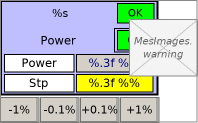
VISUALIZATION VISU_CANON  // 198x123
VAR_IN_OUT
	m_Input_SOURCE : BLOCK_SOURCE_JOULE;
END_VAR
    Rectangle (0,0 158x95)
    Rectangle (3,30 110x21), "Power"
    Rectangle (117,3 37x20), "NOK", invisible if: NOT m_Input_SOURCE.STATE_NOK
    Rectangle (117,30 37x20), "OFF", invisible if: m_Input_SOURCE.STATE_EJ_ON
    Rectangle (117,3 37x20), "OK", invisible if: m_Input_SOURCE.STATE_NOK
    Rectangle (117,30 37x20), "ON", invisible if: NOT m_Input_SOURCE.STATE_EJ_ON
    RoundedRectangle (4,54 70x18), "Power", invisible if: Global_Variables.MACHINE.State_manu
    RoundedRectangle (76,54 77x18), "%.3f %%", text variable: m_Input_SOURCE.STATE_POWER, invisible if: Global_Variables.MACHINE.State_manu
    Rectangle (0,3 120x21), "%s", text variable: m_Input_SOURCE.MNEMO
    Polyline (7,35)
    RoundedRectangle (4,74 70x18), "Stp", invisible if: NOT Global_Variables.PRG_USER.ACTU_USER.MAINTENANCE OR NOT MACHINE.State_manu
    RoundedRectangle (76,74 77x18), "%.3f %%", text variable: m_Input_SOURCE.PRM_POWER, invisible if: NOT Global_Variables.PRG_USER.ACTU_USER.MAINTENANCE OR NOT MACHINE.STATE_Manu
        OnMouseDown: write the text variable via InputWithLimits, min 0, max 100
    Rectangle (114,28 41x24), invisible if: NOT m_Input_SOURCE.EJ.AUTOR_ON_IHM AND NOT m_Input_SOURCE.EJ.AUTOR_Off_IHM, input disabled if: (NOT m_Input_SOURCE.EJ.AUTOR_ON_IHM AND NOT m_Input_SOURCE.EJ.AUTOR_OFF_IHM) OR NOT PRG_User.ACTU_USER.MAINTENANCE
        tap m_Input_SOURCE.EJ.M_On
    Image (129,19 69x57), invisible if: NOT m_Input_SOURCE.STATE_NOK, image: MesImages.warning
    Button (0,97 39x26), "-1%", invisible if: NOT Global_Variables.PRG_USER.ACTU_USER.MAINTENANCE OR NOT MACHINE.STATE_Manu OR (m_Input_SOURCE.PRM_POWER<1.0)
        OnMouseClick: execute { m_Input_SOURCE.PRM_POWER := m_Input_SOURCE.PRM_POWER - 1.0; }
    Button (40,97 39x26), "-0.1%", invisible if: NOT Global_Variables.PRG_USER.ACTU_USER.MAINTENANCE OR NOT MACHINE.STATE_Manu OR (m_Input_SOURCE.PRM_POWER<0.1)
        OnMouseClick: execute { m_Input_SOURCE.PRM_POWER := m_Input_SOURCE.PRM_POWER - 0.1; }
    Button (80,97 39x26), "+0.1%", invisible if: NOT Global_Variables.PRG_USER.ACTU_USER.MAINTENANCE OR NOT MACHINE.STATE_Manu OR (m_Input_SOURCE.PRM_POWER>99.9)
        OnMouseClick: execute { m_Input_SOURCE.PRM_POWER := m_Input_SOURCE.PRM_POWER + 0.1; }
    Button (120,97 39x26), "+1%", invisible if: NOT Global_Variables.PRG_USER.ACTU_USER.MAINTENANCE OR NOT MACHINE.STATE_Manu OR (m_Input_SOURCE.PRM_POWER>99.0)
        OnMouseClick: execute { m_Input_SOURCE.PRM_POWER := m_Input_SOURCE.PRM_POWER + 1.0; }
END_VISUALIZATION

// ---- Visualizations/Symbole/EVAP/VISU_CANON_GENIUS_ETH.TcVIS
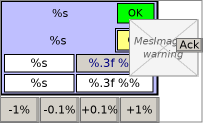
VISUALIZATION VISU_CANON_GENIUS_ETH  // 203x123
VAR_IN_OUT
	m_Input_SOURCE : BLOCK_SOURCE_GENIUS_ETHERCAT;
END_VAR
    Rectangle (0,0 158x95)
    Rectangle (3,30 110x21), "%s", text list: 'TextList_Evap', text index: 2
    Rectangle (117,3 37x20), "NOK", invisible if: NOT m_Input_SOURCE.STATE_NOK
    Rectangle (117,30 37x20), "OFF", invisible if: m_Input_SOURCE.STATE_SRC OR m_Input_SOURCE.STATE_SRC_ON
    Rectangle (117,3 37x20), "OK", invisible if: m_Input_SOURCE.STATE_NOK
    Rectangle (117,30 37x20), "ON", invisible if: NOT m_Input_SOURCE.STATE_SRC AND NOT m_Input_SOURCE.STATE_SRC_ON
    RoundedRectangle (4,54 70x18), "%s", invisible if: Global_Variables.MACHINE.State_manu, text list: 'TextList_Evap', text index: 4
    RoundedRectangle (76,54 77x18), "%.3f %%", text variable: m_Input_SOURCE.STATE_COURANT, invisible if: Global_Variables.MACHINE.State_manu
    Rectangle (117,30 37x20), "ON", invisible if: m_Input_SOURCE.STATE_SRC_ON OR NOT m_Input_SOURCE.STATE_SRC
    Rectangle (0,3 120x21), "%s", text variable: m_Input_SOURCE.MNEMO
    Polyline (7,35)
    RoundedRectangle (4,74 70x18), "%s", invisible if: NOT Global_Variables.PRG_USER.ACTU_USER.MAINTENANCE OR NOT MACHINE.State_manu, text list: 'TextList_Evap', text index: 4
    RoundedRectangle (76,74 77x18), "%.3f %%", text variable: m_Input_SOURCE.PRM_COURANT, invisible if: NOT Global_Variables.PRG_USER.ACTU_USER.MAINTENANCE OR NOT MACHINE.STATE_Manu
        OnMouseDown: write the text variable via VisuDialogs.Numpad, min 0, max 100
    Rectangle (115,28 41x24), invisible if: NOT m_Input_SOURCE.SRC.AUTOR_ON_IHM AND NOT m_Input_SOURCE.SRC.AUTOR_OFF_IHM, input disabled if: (NOT m_Input_SOURCE.SRC.AUTOR_ON_IHM AND NOT m_Input_SOURCE.SRC.AUTOR_OFF_IHM) OR NOT PRG_User.ACTU_USER.MAINTENANCE
        tap m_Input_SOURCE.SRC.M_On
    Image (129,19 69x57), invisible if: NOT m_Input_SOURCE.SRC.STATE_Nok AND NOT m_Input_SOURCE.DEF_Source.DEF AND NOT m_Input_SOURCE.DEF_Communication.DEF, image: MesImages.warning
    Button (0,97 39x26), "-1%", invisible if: NOT Global_Variables.PRG_USER.ACTU_USER.MAINTENANCE OR NOT MACHINE.STATE_Manu
        OnMouseClick: execute { m_Input_SOURCE.PRM_COURANT := m_Input_SOURCE.PRM_COURANT - 1; }
    Button (40,97 39x26), "-0.1%", invisible if: NOT Global_Variables.PRG_USER.ACTU_USER.MAINTENANCE OR NOT MACHINE.STATE_Manu
        OnMouseClick: execute { m_Input_SOURCE.PRM_COURANT := m_Input_SOURCE.PRM_COURANT - 0.1; }
    Button (80,97 39x26), "+0.1%", invisible if: NOT Global_Variables.PRG_USER.ACTU_USER.MAINTENANCE OR NOT MACHINE.STATE_Manu
        OnMouseClick: execute { m_Input_SOURCE.PRM_COURANT := m_Input_SOURCE.PRM_COURANT + 0.1; }
    Button (120,97 39x26), "+1%", invisible if: NOT Global_Variables.PRG_USER.ACTU_USER.MAINTENANCE OR NOT MACHINE.STATE_Manu
        OnMouseClick: execute { m_Input_SOURCE.PRM_COURANT := m_Input_SOURCE.PRM_COURANT + 1; }
    Button (176,38 27x14), "Ack", invisible if: NOT m_Input_SOURCE.HV.STATE_Nok AND NOT m_Input_SOURCE.DEF_Source.DEF AND NOT m_Input_SOURCE.DEF_Communication.DEF AND NOT m_Input_SOURCE.DEF_HV.DEF
        tap m_Input_SOURCE.M_Ack
END_VISUALIZATION

// ---- Visualizations/Symbole/EVAP/VISU_CANON_ST10.TcVIS
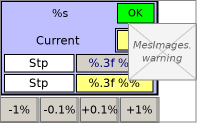
VISUALIZATION VISU_CANON_ST10  // 197x123
VAR_IN_OUT
	m_Input_SOURCE : BLOCK_CANON_ST10;
END_VAR
    Rectangle (0,0 158x95)
    Rectangle (3,30 110x21), "Current"
    Rectangle (117,3 37x20), "NOK", invisible if: NOT m_Input_SOURCE.STATE_NOK
    Rectangle (117,30 37x20), "OFF", invisible if: m_Input_SOURCE.STATE_SRC OR m_Input_SOURCE.STATE_SRC_ON
    Rectangle (117,3 37x20), "OK", invisible if: m_Input_SOURCE.STATE_NOK
    Rectangle (117,30 37x20), "ON", invisible if: NOT m_Input_SOURCE.STATE_SRC AND NOT m_Input_SOURCE.STATE_SRC_ON
    RoundedRectangle (4,54 70x18), "Stp", invisible if: Global_Variables.MACHINE.State_manu
    RoundedRectangle (76,54 77x18), "%.3f %%", text variable: m_Input_SOURCE.AO_QIEM.Value, invisible if: Global_Variables.MACHINE.State_manu
    Rectangle (117,30 37x20), "ON", invisible if: m_Input_SOURCE.STATE_SRC_ON OR Not m_Input_SOURCE.STATE_SRC
    Rectangle (0,3 120x21), "%s", text variable: m_Input_SOURCE.MNEMO
    Polyline (7,35)
    RoundedRectangle (4,74 70x18), "Stp", invisible if: NOT Global_Variables.PRG_USER.ACTU_USER.MAINTENANCE OR NOT MACHINE.State_manu
    RoundedRectangle (76,74 77x18), "%.3f %%", text variable: m_Input_SOURCE.PRM_COURANT, invisible if: NOT Global_Variables.PRG_USER.ACTU_USER.MAINTENANCE OR NOT MACHINE.STATE_Manu
        OnMouseDown: write the text variable via InputWithLimits, min 0, max 100
    Rectangle (115,28 41x24), invisible if: NOT m_Input_SOURCE.SRC.AUTOR_ON_IHM AND NOT m_Input_SOURCE.SRC.AUTOR_OFF_IHM, input disabled if: (NOT m_Input_SOURCE.SRC.AUTOR_ON_IHM AND NOT m_Input_SOURCE.SRC.AUTOR_OFF_IHM) OR NOT PRG_User.ACTU_USER.MAINTENANCE
        tap m_Input_SOURCE.SRC.M_On
    Image (128,23 69x57), invisible if: NOT m_Input_SOURCE.STATE_NOK, image: MesImages.warning
    Button (0,97 39x26), "-1%", invisible if: NOT Global_Variables.PRG_USER.ACTU_USER.MAINTENANCE OR NOT MACHINE.STATE_Manu OR (m_Input_SOURCE.PRM_COURANT<1.0)
        OnMouseClick: execute { m_Input_SOURCE.PRM_COURANT := m_Input_SOURCE.PRM_COURANT - 1.0; }
    Button (40,97 39x26), "-0.1%", invisible if: NOT Global_Variables.PRG_USER.ACTU_USER.MAINTENANCE OR NOT MACHINE.STATE_Manu OR (m_Input_SOURCE.PRM_COURANT<0.1)
        OnMouseClick: execute { m_Input_SOURCE.PRM_COURANT := m_Input_SOURCE.PRM_COURANT - 0.1; }
    Button (80,97 39x26), "+0.1%", invisible if: NOT Global_Variables.PRG_USER.ACTU_USER.MAINTENANCE OR NOT MACHINE.STATE_Manu OR (m_Input_SOURCE.PRM_COURANT>99.9)
        OnMouseClick: execute { m_Input_SOURCE.PRM_COURANT := m_Input_SOURCE.PRM_COURANT + 0.1; }
    Button (120,97 39x26), "+1%", invisible if: NOT Global_Variables.PRG_USER.ACTU_USER.MAINTENANCE OR NOT MACHINE.STATE_Manu OR (m_Input_SOURCE.PRM_COURANT>99.0)
        OnMouseClick: execute { m_Input_SOURCE.PRM_COURANT := m_Input_SOURCE.PRM_COURANT + 1.0; }
END_VISUALIZATION

// ---- Visualizations/Symbole/EVAP/VISU_CONF_BAL.TcVIS
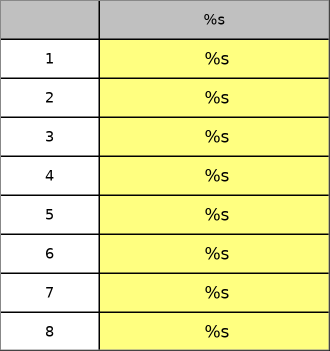
VISUALIZATION VISU_CONF_BAL  // 330x351
VAR_IN_OUT
	m_Input_SWEEP : BLOCK_TELEMARK_CHEETAH_SWEEP;
END_VAR
    Rectangle (0,0 99x39)
    Rectangle (99,39 231x39), "%s", text variable: m_Input_SWEEP.PRM_BAL[1], input disabled if: NOT Global_Variables.PRG_USER.ACTU_USER.CONF_MACHINE
        OnMouseDown: write the text variable via InputWithLimits
    Rectangle (99,0 231x39), "%s", text list: 'TextList_Config_Evap', text index: 8
    Rectangle (0,39 99x39), "1"
    Rectangle (0,78 99x39), "2"
    Rectangle (99,78 231x39), "%s", text variable: m_Input_SWEEP.PRM_BAL[2], input disabled if: NOT Global_Variables.PRG_USER.ACTU_USER.CONF_MACHINE
        OnMouseDown: write the text variable via InputWithLimits
    Rectangle (0,117 99x39), "3"
    Rectangle (99,117 231x39), "%s", text variable: m_Input_SWEEP.PRM_BAL[3], input disabled if: NOT Global_Variables.PRG_USER.ACTU_USER.CONF_MACHINE
        OnMouseDown: write the text variable via InputWithLimits
    Rectangle (0,156 99x39), "4"
    Rectangle (99,156 231x39), "%s", text variable: m_Input_SWEEP.PRM_BAL[4], input disabled if: NOT Global_Variables.PRG_USER.ACTU_USER.CONF_MACHINE
        OnMouseDown: write the text variable via InputWithLimits
    Rectangle (99,195 231x39), "%s", text variable: m_Input_SWEEP.PRM_BAL[5], input disabled if: NOT Global_Variables.PRG_USER.ACTU_USER.CONF_MACHINE
        OnMouseDown: write the text variable via InputWithLimits
    Rectangle (0,195 99x39), "5"
    Rectangle (0,234 99x39), "6"
    Rectangle (99,234 231x39), "%s", text variable: m_Input_SWEEP.PRM_BAL[6], input disabled if: NOT Global_Variables.PRG_USER.ACTU_USER.CONF_MACHINE
        OnMouseDown: write the text variable via InputWithLimits
    Rectangle (0,273 99x39), "7"
    Rectangle (99,273 231x39), "%s", text variable: m_Input_SWEEP.PRM_BAL[7], input disabled if: NOT Global_Variables.PRG_USER.ACTU_USER.CONF_MACHINE
        OnMouseDown: write the text variable via InputWithLimits
    Rectangle (0,312 99x39), "8"
    Rectangle (99,312 231x39), "%s", text variable: m_Input_SWEEP.PRM_BAL[8], input disabled if: NOT Global_Variables.PRG_USER.ACTU_USER.CONF_MACHINE
        OnMouseDown: write the text variable via InputWithLimits
END_VISUALIZATION

// ---- Visualizations/Symbole/EVAP/VISU_CONF_MAT.TcVIS
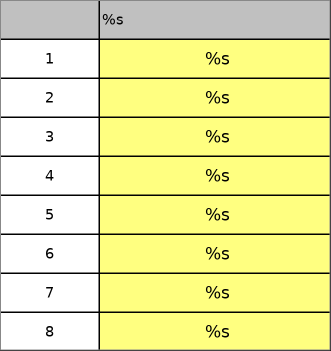
VISUALIZATION VISU_CONF_MAT  // 331x351
VAR_IN_OUT
	m_Input_CRUCIBLE : BLOCK_IND_CR_396_TELEMARK;
END_VAR
    Rectangle (0,0 99x39)
    Rectangle (99,39 232x39), "%s", text variable: m_Input_CRUCIBLE.PRM_MAT[1], input disabled if: NOT Global_Variables.PRG_USER.ACTU_USER.CONF_MACHINE
        OnMouseDown: write the text variable via InputWithLimits
    Rectangle (99,0 232x39), "%s", text list: 'TextList_Config_Evap', text index: 7
    Rectangle (0,39 99x39), "1"
    Rectangle (0,78 99x39), "2", invisible if: m_Input_CRUCIBLE.CONF_NCR <2
    Rectangle (99,78 232x39), "%s", text variable: m_Input_CRUCIBLE.PRM_MAT[2], invisible if: m_Input_CRUCIBLE.CONF_NCR <2, input disabled if: NOT Global_Variables.PRG_USER.ACTU_USER.CONF_MACHINE
        OnMouseDown: write the text variable via InputWithLimits
    Rectangle (0,117 99x39), "3", invisible if: m_Input_CRUCIBLE.CONF_NCR <3
    Rectangle (99,117 232x39), "%s", text variable: m_Input_CRUCIBLE.PRM_MAT[3], invisible if: m_Input_CRUCIBLE.CONF_NCR <3, input disabled if: NOT Global_Variables.PRG_USER.ACTU_USER.CONF_MACHINE
        OnMouseDown: write the text variable via InputWithLimits
    Rectangle (0,156 99x39), "4", invisible if: m_Input_CRUCIBLE.CONF_NCR <4
    Rectangle (99,156 232x39), "%s", text variable: m_Input_CRUCIBLE.PRM_MAT[4], invisible if: m_Input_CRUCIBLE.CONF_NCR <4, input disabled if: NOT Global_Variables.PRG_USER.ACTU_USER.CONF_MACHINE
        OnMouseDown: write the text variable via InputWithLimits
    Rectangle (0,195 99x39), "5", invisible if: m_Input_CRUCIBLE.CONF_NCR <5
    Rectangle (99,195 232x39), "%s", text variable: m_Input_CRUCIBLE.PRM_MAT[5], invisible if: m_Input_CRUCIBLE.CONF_NCR <5, input disabled if: NOT Global_Variables.PRG_USER.ACTU_USER.CONF_MACHINE
        OnMouseDown: write the text variable via InputWithLimits
    Rectangle (0,234 99x39), "6", invisible if: m_Input_CRUCIBLE.CONF_NCR <6
    Rectangle (99,234 232x39), "%s", text variable: m_Input_CRUCIBLE.PRM_MAT[6], invisible if: m_Input_CRUCIBLE.CONF_NCR <6, input disabled if: NOT Global_Variables.PRG_USER.ACTU_USER.CONF_MACHINE
        OnMouseDown: write the text variable via InputWithLimits
    Rectangle (0,273 99x39), "7", invisible if: m_Input_CRUCIBLE.CONF_NCR <7
    Rectangle (99,273 232x39), "%s", text variable: m_Input_CRUCIBLE.PRM_MAT[7], invisible if: m_Input_CRUCIBLE.CONF_NCR <7, input disabled if: NOT Global_Variables.PRG_USER.ACTU_USER.CONF_MACHINE
        OnMouseDown: write the text variable via InputWithLimits
    Rectangle (0,312 99x39), "8", invisible if: m_Input_CRUCIBLE.CONF_NCR <8
    Rectangle (99,312 232x39), "%s", text variable: m_Input_CRUCIBLE.PRM_MAT[8], invisible if: m_Input_CRUCIBLE.CONF_NCR <8, input disabled if: NOT Global_Variables.PRG_USER.ACTU_USER.CONF_MACHINE
        OnMouseDown: write the text variable via InputWithLimits
END_VISUALIZATION

// ---- Visualizations/Symbole/EVAP/VISU_CREUSET_old.TcVIS
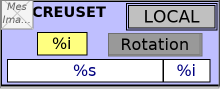
VISUALIZATION VISU_CREUSET_old  // 220x89
VAR_IN_OUT
	m_Input_CREUSET : BLOCK_IND_CR_379_TELEMARK;
END_VAR
    Rectangle (0,0 220x86)
    RoundedRectangle (37,32 50x23), "%i", text variable: m_Input_CREUSET.PRM_NCR, invisible if: NOT Global_Variables.PRG_USER.ACTU_USER.MAINTENANCE OR NOT MACHINE.State_manu
        OnMouseDown: write the text variable via InputWithLimits, min 1, max m_Input_CREUSET.CONF_NCR
    Rectangle (6,3 126x18), "CREUSET"
    RoundedRectangle (7,59 156x23), "%s", text variable: m_Input_CREUSET.STATE_MAT
    RoundedRectangle (163,59 47x23), "%i", text variable: m_Input_CREUSET.STATE_POS
    Button (108,33 94x23), "Rotation", invisible if: NOT m_Input_CREUSET.AUTOR_Change_IHM OR NOT PRG_User.ACTU_USER.MAINTENANCE
        tap m_Input_CREUSET.M_Change
    Image (1,-3 32x32), invisible if: NOT m_Input_CREUSET.State_nok, image: MesImages.warning
    RoundedRectangle (128,5 87x23), "REMOTE", invisible if: not m_Input_CREUSET.OUT_RMT
    RoundedRectangle (128,5 87x23), "LOCAL", invisible if: m_Input_CREUSET.OUT_RMT
    Rectangle (126,3 91x27), invisible if: Not m_Input_CREUSET.AUTOR_Remote_IHM, input disabled if: NOT PRG_User.ACTU_USER.MAINTENANCE
        tap m_Input_CREUSET.M_Remote
END_VISUALIZATION

// ---- Visualizations/Symbole/EVAP/VISU_CREUSET.TcVIS
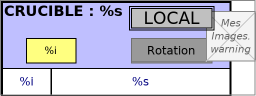
VISUALIZATION VISU_CREUSET  // 256x96
VAR_IN_OUT
	m_Input_CREUSET : BLOCK_IND_CR_396_TELEMARK;
END_VAR
VAR_INPUT
	m_Input_NUM_CRUCIBLE : SINT;
END_VAR
    Rectangle (1,1 230x95), "CRUCIBLE : %s", text variable: m_Input_NUM_CRUCIBLE
    RoundedRectangle (26,38 50x25), "%i", text variable: m_Input_CREUSET.PRM_NCR, invisible if: NOT Global_Variables.PRG_USER.ACTU_USER.MAINTENANCE OR NOT MACHINE.State_manu
        OnMouseDown: write the text variable via InputWithLimits, min 1, max 6
    Rectangle (51,68 179x27), "%s", text variable: m_Input_CREUSET.STATE_MAT
    Rectangle (2,68 49x27), "%i", text variable: m_Input_CREUSET.STATE_POS
    Button (131,38 81x25), "Rotation", colour toggle: m_Input_CREUSET.STATE_ROT, invisible if: NOT m_Input_CREUSET.AUTOR_Change_IHM OR NOT PRG_User.ACTU_USER.MAINTENANCE
        tap m_Input_CREUSET.M_Change
    Image (206,11 50x50), invisible if: NOT m_Input_CREUSET.State_nok, image: MesImages.warning
    RoundedRectangle (131,8 81x20), "REMOTE", invisible if: not m_Input_CREUSET.OUT_RMT
    RoundedRectangle (131,8 81x20), "LOCAL", invisible if: m_Input_CREUSET.OUT_RMT
    Rectangle (129,6 85x24), invisible if: Not m_Input_CREUSET.AUTOR_Remote_IHM, input disabled if: NOT PRG_User.ACTU_USER.MAINTENANCE
        tap m_Input_CREUSET.M_Remote
END_VISUALIZATION

// ---- Visualizations/Symbole/EVAP/VISU_CREUSET_V3.TcVIS
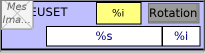
VISUALIZATION VISU_CREUSET_V3  // 205x53
VAR_IN_OUT
	m_Input_CREUSET : BLOCK_IND_CR_379_TELEMARK_V3;
END_VAR
    Rectangle (0,0 205x50)
    RoundedRectangle (96,2 45x22), "%i", text variable: m_Input_CREUSET.PRM_NCR, invisible if: NOT Global_Variables.PRG_USER.ACTU_USER.MAINTENANCE OR NOT MACHINE.State_manu
        OnMouseDown: write the text variable via InputWithLimits
    Rectangle (0,3 81x18), "CREUSET"
    Rectangle (1,26 48x18), text list: 'TextList_Evap', text index: 5
    RoundedRectangle (46,26 116x20), "%s", text variable: m_Input_CREUSET.STATE_MAT
    RoundedRectangle (162,26 38x20), "%i", text variable: m_Input_CREUSET.STATE_POS
    Button (148,3 51x20), "Rotation", invisible if: NOT m_Input_CREUSET.AUTOR_Change_IHM OR NOT PRG_User.ACTU_USER.MAINTENANCE
        tap m_Input_CREUSET.M_Change
    Image (1,-3 32x32), invisible if: NOT m_Input_CREUSET.State_nok, image: MesImages.warning
END_VISUALIZATION

// ---- Visualizations/Symbole/EVAP/VISU_CR_SW_GENIUS_ETH.TcVIS
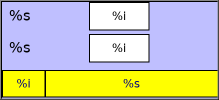
VISUALIZATION VISU_CR_SW_GENIUS_ETH  // 219x100
VAR_IN_OUT
	m_Input_BALAYAGE : BLOCK_IND_CREUSET_GENIUS_ETHERCAT;
END_VAR
    Rectangle (0,0 219x100)
    Rectangle (6,1 118x29), "%s", text list: 'TextList_Evap', text index: 0
    Rectangle (2,70 43x27), "%i", text variable: m_Input_BALAYAGE.STATE_POS_CR
    Rectangle (45,70 173x27), "%s", text variable: m_Input_BALAYAGE.STATE_MAT
    RoundedRectangle (89,2 60x28), "%i", text variable: m_Input_BALAYAGE.PRM_NCR, input disabled if: NOT Global_Variables.PRG_USER.ACTU_USER.MAINTENANCE OR NOT MACHINE.STATE_Manu
        OnMouseDown: write the text variable via VisuDialogs.Numpad, min 1, max m_Input_BALAYAGE.CONF_NCR
    Rectangle (6,33 118x29), "%s", text list: 'TextList_Evap', text index: 1
    RoundedRectangle (89,34 60x28), "%i", text variable: m_Input_BALAYAGE.PRM_NBAL, input disabled if: NOT Global_Variables.PRG_USER.ACTU_USER.MAINTENANCE OR NOT MACHINE.STATE_Manu
        OnMouseDown: write the text variable via VisuDialogs.Numpad, min 1, max 8
END_VISUALIZATION

// ---- Visualizations/Symbole/EVAP/VISU_HT_CANON_ST10.TcVIS
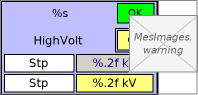
VISUALIZATION VISU_HT_CANON_ST10  // 198x95
VAR_IN_OUT
	m_Input_SOURCE : BLOCK_CANON_ST10;
END_VAR
    Rectangle (0,0 158x95)
    Rectangle (3,30 110x21), "HighVolt"
    Rectangle (117,3 37x20), "NOK", invisible if: NOT m_Input_SOURCE.STATE_NOK
    Rectangle (117,30 37x20), "OFF", invisible if: m_Input_SOURCE.STATE_HV OR m_Input_SOURCE.STATE_HV_ON
    Rectangle (117,3 37x20), "OK", invisible if: m_Input_SOURCE.STATE_NOK
    Rectangle (117,30 37x20), "ON", invisible if: NOT m_Input_SOURCE.STATE_HV AND NOT m_Input_SOURCE.STATE_HV_ON
    RoundedRectangle (4,54 70x18), "Stp", invisible if: Global_Variables.MACHINE.State_manu
    RoundedRectangle (76,54 77x18), "%.2f kV", text variable: m_Input_SOURCE.AO_QUHV.Value, invisible if: Global_Variables.MACHINE.State_manu
    Rectangle (117,30 37x20), "ON", invisible if: m_Input_SOURCE.STATE_HV_ON OR NOT m_Input_SOURCE.STATE_HV
    Rectangle (0,3 120x21), "%s", text variable: m_Input_SOURCE.MNEMO
    Polyline (7,35)
    RoundedRectangle (4,74 70x18), "Stp", invisible if: NOT Global_Variables.PRG_USER.ACTU_USER.MAINTENANCE OR NOT MACHINE.State_manu
    RoundedRectangle (76,74 77x18), "%.2f kV", text variable: m_Input_SOURCE.PRM_TENSION, invisible if: NOT Global_Variables.PRG_USER.ACTU_USER.MAINTENANCE OR NOT MACHINE.STATE_Manu
        OnMouseDown: write the text variable via InputWithLimits, min 7, max 10
    Rectangle (115,28 41x24), invisible if: NOT m_Input_SOURCE.HV.AUTOR_ON_IHM AND NOT m_Input_SOURCE.HV.AUTOR_OFF_IHM, input disabled if: (NOT m_Input_SOURCE.HV.AUTOR_ON_IHM AND NOT m_Input_SOURCE.HV.AUTOR_OFF_IHM) OR NOT PRG_User.ACTU_USER.MAINTENANCE
        tap m_Input_SOURCE.HV.M_On
    Image (129,15 69x57), invisible if: NOT m_Input_SOURCE.STATE_NOK, image: MesImages.warning
END_VISUALIZATION

// ---- Visualizations/Symbole/EVAP/VISU_HT_GENIUS_ETH.TcVIS
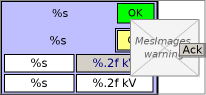
VISUALIZATION VISU_HT_GENIUS_ETH  // 206x95
VAR_IN_OUT
	m_Input_SOURCE : BLOCK_SOURCE_GENIUS_ETHERCAT;
END_VAR
    Rectangle (0,0 158x95)
    Rectangle (3,30 110x21), "%s", text list: 'TextList_Evap', text index: 3
    Rectangle (117,3 37x20), "NOK", invisible if: NOT m_Input_SOURCE.STATE_NOK
    Rectangle (117,30 37x20), "OFF", invisible if: m_Input_SOURCE.STATE_HV OR m_Input_SOURCE.STATE_HV_ON
    Rectangle (117,3 37x20), "OK", invisible if: m_Input_SOURCE.STATE_NOK
    Rectangle (117,30 37x20), "ON", invisible if: NOT m_Input_SOURCE.STATE_HV AND NOT m_Input_SOURCE.STATE_HV_ON
    RoundedRectangle (4,54 70x18), "%s", invisible if: Global_Variables.MACHINE.State_manu, text list: 'TextList_Evap', text index: 4
    RoundedRectangle (76,54 77x18), "%.2f kV", text variable: m_Input_SOURCE.STATE_TENSION, invisible if: Global_Variables.MACHINE.State_manu
    Rectangle (117,30 37x20), "ON", invisible if: m_Input_SOURCE.STATE_HV_ON OR NOT m_Input_SOURCE.STATE_HV
    Rectangle (0,3 120x21), "%s", text variable: m_Input_SOURCE.MNEMO
    Polyline (7,35)
    RoundedRectangle (4,74 70x18), "%s", invisible if: NOT Global_Variables.PRG_USER.ACTU_USER.MAINTENANCE OR NOT MACHINE.State_manu, text list: 'TextList_Evap', text index: 4
    RoundedRectangle (76,74 77x18), "%.2f kV", text variable: m_Input_SOURCE.PRM_TENSION, invisible if: NOT Global_Variables.PRG_USER.ACTU_USER.MAINTENANCE OR NOT MACHINE.STATE_Manu
        OnMouseDown: write the text variable via VisuDialogs.Numpad, min 7, max 10
    Rectangle (115,28 41x24), invisible if: NOT m_Input_SOURCE.HV.AUTOR_ON_IHM AND NOT m_Input_SOURCE.HV.AUTOR_OFF_IHM, input disabled if: (NOT m_Input_SOURCE.HV.AUTOR_ON_IHM AND NOT m_Input_SOURCE.HV.AUTOR_OFF_IHM) OR NOT PRG_User.ACTU_USER.MAINTENANCE
        tap m_Input_SOURCE.HV.M_On
    Image (130,19 69x57), invisible if: NOT m_Input_SOURCE.HV.STATE_Nok AND NOT m_Input_SOURCE.DEF_Source.DEF AND NOT m_Input_SOURCE.DEF_Communication.DEF AND NOT m_Input_SOURCE.DEF_HV.DEF, image: MesImages.warning
    Button (179,43 27x14), "Ack", invisible if: NOT m_Input_SOURCE.HV.STATE_Nok AND NOT m_Input_SOURCE.DEF_Source.DEF AND NOT m_Input_SOURCE.DEF_Communication.DEF AND NOT m_Input_SOURCE.DEF_HV.DEF
        tap m_Input_SOURCE.M_Ack
END_VISUALIZATION

// ---- Visualizations/Symbole/EVAP/VISU_SOURCE_EFFET_JOULE.TcVIS
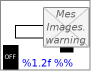
VISUALIZATION VISU_SOURCE_EFFET_JOULE  // 91x71
VAR_IN_OUT
	m_Input_SOURCE : BLOCK_SOURCE_JOULE;
END_VAR
    Polygon (30,49)
    Rectangle (15,57 65x12), "%1.2f %%", text variable: m_Input_SOURCE.STATE_POWER
    Polyline (69,38)
    Polyline (20,37)
    Rectangle (15,25 48x13)
    Polyline (65,41), colour toggle: m_Input_SOURCE.EJ.STATE_ON
    Rectangle (4,45 13x22), "ON", invisible if: NOT m_Input_SOURCE.STATE_EJ_ON
    Rectangle (4,46 13x22), "OFF", invisible if: m_Input_SOURCE.STATE_EJ_ON
    Rectangle (3,45 15x24), invisible if: NOT m_Input_SOURCE.EJ.AUTOR_ON_IHM AND NOT m_Input_SOURCE.EJ.AUTOR_OFF_IHM, input disabled if: (NOT m_Input_SOURCE.EJ.AUTOR_ON_IHM AND NOT m_Input_SOURCE.EJ.AUTOR_OFF_IHM) OR NOT PRG_User.ACTU_USER.MAINTENANCE
        tap m_Input_SOURCE.EJ.M_On
    Polygon (45,28), invisible if: NOT ( m_Input_SOURCE.EJ.STATE_On AND (m_Input_SOURCE.STATE_power > 0) )
    Rectangle (60,47 13x5), colour toggle: m_Input_SOURCE.WATER
    Image (43,7 46x40), invisible if: NOT m_Input_SOURCE.STATE_NOK, image: MesImages.warning
END_VISUALIZATION

// ---- Visualizations/Symbole/EVAP/VISU_SOURCE_EVAP_COTE_GENIUS_ETH.TcVIS
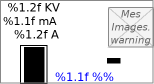
VISUALIZATION VISU_SOURCE_EVAP_COTE_GENIUS_ETH  // 154x84
VAR_IN_OUT
	m_Input_SOURCE : BLOCK_SOURCE_GENIUS_ETHERCAT;
END_VAR
VAR_INPUT
	m_Input_NO_IFIL_RET : BOOL;
	m_Input_NO_HV_RET : BOOL;
	m_Input_NO_IEMISS_RET : BOOL;
END_VAR
    Polygon (84,73), colour toggle: m_Input_SOURCE.STATE_SRC_ON, invisible if: NOT m_Input_SOURCE.STATE_SRC_ON AND NOT m_Input_SOURCE.STATE_SRC
    Polygon (84,71), invisible if: m_Input_SOURCE.STATE_SRC_ON OR (m_Input_SOURCE.STATE_SRC OR m_Input_SOURCE.STATE_SRC)
    Polygon (70,46)
    Polygon (84,43), invisible if: NOT (m_Input_SOURCE.SRC.STATE_On AND m_Input_SOURCE.HV.STATE_On AND (m_Input_SOURCE.STATE_I_EMISS>0.0))
    Rectangle (1,15 62x13), "%1.1f mA", text variable: m_Input_SOURCE.STATE_I_EMISS, invisible if: m_Input_NO_IEMISS_RET
    Rectangle (45,70 79x14), "%1.1f %%", text variable: m_Input_SOURCE.STATE_COURANT
    Rectangle (47,46 77x37), invisible if: (NOT m_Input_SOURCE.SRC.AUTOR_ON_IHM AND NOT m_Input_SOURCE.SRC.AUTOR_OFF_IHM) OR NOT PRG_User.ACTU_USER.MAINTENANCE, input disabled if: (NOT m_Input_SOURCE.SRC.AUTOR_ON_IHM AND NOT m_Input_SOURCE.SRC.AUTOR_OFF_IHM) OR NOT PRG_User.ACTU_USER.MAINTENANCE
        OnMouseUp: execute { m_Input_SOURCE.SRC.M_On:=(TRUE); }
    Rectangle (107,58 13x5), colour toggle: m_Input_SOURCE.WATER
    Rectangle (3,28 59x13), "%1.2f A", text variable: m_Input_SOURCE.STATE_I_Fil, invisible if: m_Input_NO_IFIL_RET
    Image (108,7 46x40), invisible if: NOT m_Input_SOURCE.STATE_NOK, image: MesImages.warning
    Rectangle (1,1 62x13), "%1.2f KV", text variable: m_Input_SOURCE.STATE_V_HV, invisible if: m_Input_NO_HV_RET
    Rectangle (24,47 20x34), colour toggle: (m_Input_SOURCE.STATE_HV_ON), invisible if: NOT m_Input_SOURCE.STATE_HV_ON AND NOT m_Input_SOURCE.STATE_HV
    Rectangle (24,47 20x35), invisible if: (m_Input_SOURCE.STATE_HV_ON OR m_Input_SOURCE.STATE_HV)
    Polygon (41,73)
    Rectangle (20,45 27x39), invisible if: NOT m_Input_SOURCE.HV.AUTOR_ON_IHM AND NOT m_Input_SOURCE.HV.AUTOR_OFF_IHM, input disabled if: (NOT m_Input_SOURCE.HV.AUTOR_ON_IHM AND NOT m_Input_SOURCE.HV.AUTOR_OFF_IHM) OR NOT PRG_User.ACTU_USER.MAINTENANCE
        OnMouseUp: execute { m_Input_SOURCE.HV.M_On:=(TRUE); }
END_VISUALIZATION

// ---- Visualizations/Symbole/EVAP/VISU_SOURCE_EVAP_COTE_ST10.TcVIS
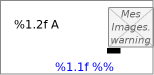
VISUALIZATION VISU_SOURCE_EVAP_COTE_ST10  // 154x75
VAR_IN_OUT
	m_Input_SOURCE : BLOCK_CANON_ST10;
END_VAR
VAR_INPUT
	m_Input_NO_IFIL_RET : Bool;
END_VAR
VAR_INPUT
	m_Input_NO_IEMISS_RET : Bool;
END_VAR
    Polygon (84,73), colour toggle: m_Input_SOURCE.STATE_SRC_ON, invisible if: NOT m_Input_SOURCE.STATE_SRC_ON AND NOT m_Input_SOURCE.STATE_SRC
    Polygon (84,71), invisible if: m_Input_SOURCE.STATE_SRC_ON OR (m_Input_SOURCE.STATE_SRC OR m_Input_SOURCE.STATE_SRC)
    Polygon (70,46)
    Polygon (84,43), invisible if: NOT (m_Input_SOURCE.SRC.STATE_On AND m_Input_SOURCE.HV.STATE_On AND (m_Input_SOURCE.STATE_COURANT>0.0))
    Rectangle (45,60 79x14), "%1.1f %%", text variable: m_Input_SOURCE.STATE_COURANT
    Rectangle (45,36 79x39), invisible if: (NOT m_Input_SOURCE.SRC.AUTOR_ON_IHM AND NOT m_Input_SOURCE.SRC.AUTOR_OFF_IHM) OR NOT PRG_User.ACTU_USER.MAINTENANCE, input disabled if: (NOT m_Input_SOURCE.SRC.AUTOR_ON_IHM AND NOT m_Input_SOURCE.SRC.AUTOR_OFF_IHM) OR NOT PRG_User.ACTU_USER.MAINTENANCE
        OnMouseUp: execute { m_Input_SOURCE.SRC.M_On:=(TRUE); }
    Rectangle (107,48 13x5), colour toggle: m_Input_SOURCE.WATER
    Rectangle (3,18 59x13), "%1.2f A", text variable: m_Input_SOURCE.STATE_I_Fil, invisible if: m_Input_NO_IFIL_RET
    Image (108,7 46x40), invisible if: NOT m_Input_SOURCE.STATE_NOK, image: MesImages.warning
END_VISUALIZATION

// ---- Visualizations/Symbole/EVAP/VISU_SOURCE_EVAP_COTE_ST10_avec_emission.TcVIS
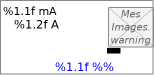
VISUALIZATION VISU_SOURCE_EVAP_COTE_ST10_avec_emission  // 154x75
VAR_IN_OUT
	m_Input_SOURCE : BLOCK_CANON_ST10;
END_VAR
VAR_INPUT
	m_Input_NO_IFIL_RET : Bool;
END_VAR
VAR_INPUT
	m_Input_NO_IEMISS_RET : Bool;
END_VAR
    Polygon (84,73), colour toggle: m_Input_SOURCE.STATE_SRC_ON, invisible if: NOT m_Input_SOURCE.STATE_SRC_ON AND NOT m_Input_SOURCE.STATE_SRC
    Polygon (84,71), invisible if: m_Input_SOURCE.STATE_SRC_ON OR (m_Input_SOURCE.STATE_SRC OR m_Input_SOURCE.STATE_SRC)
    Polygon (70,46)
    Polygon (84,43), invisible if: NOT (m_Input_SOURCE.SRC.STATE_On AND m_Input_SOURCE.HV.STATE_On AND (m_Input_SOURCE.STATE_COURANT>0.0))
    Rectangle (1,5 62x13), "%1.1f mA", text variable: m_Input_SOURCE.STATE_I_EMISS, invisible if: m_Input_NO_IEMISS_RET
    Rectangle (45,60 79x14), "%1.1f %%", text variable: m_Input_SOURCE.STATE_COURANT
    Rectangle (45,36 79x39), invisible if: (NOT m_Input_SOURCE.SRC.AUTOR_ON_IHM AND NOT m_Input_SOURCE.SRC.AUTOR_OFF_IHM) OR NOT PRG_User.ACTU_USER.MAINTENANCE, input disabled if: (NOT m_Input_SOURCE.SRC.AUTOR_ON_IHM AND NOT m_Input_SOURCE.SRC.AUTOR_OFF_IHM) OR NOT PRG_User.ACTU_USER.MAINTENANCE
        OnMouseUp: execute { m_Input_SOURCE.SRC.M_On:=(TRUE); }
    Rectangle (107,48 13x5), colour toggle: m_Input_SOURCE.WATER
    Rectangle (3,18 59x13), "%1.2f A", text variable: m_Input_SOURCE.STATE_I_Fil, invisible if: m_Input_NO_IFIL_RET
    Image (108,7 46x40), invisible if: NOT m_Input_SOURCE.STATE_NOK, image: MesImages.warning
END_VISUALIZATION

// ---- Visualizations/Symbole/EVAP/VISU_SWEEP_DIGITAL.TcVIS
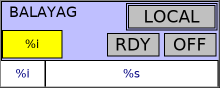
VISUALIZATION VISU_SWEEP_DIGITAL  // 220x88
VAR_IN_OUT
	m_Input_BALAYAGE : BLOCK_TELEMARK_DIGITAL_SWEEP;
END_VAR
    Rectangle (0,0 220x88)
    Rectangle (6,1 117x22), "BALAYAG"
    Rectangle (0,60 45x27), "%i", text variable: m_Input_BALAYAGE.STATE_NbBal
    Rectangle (45,60 173x27), "%s", text variable: m_Input_BALAYAGE.STATE_BAL
    RoundedRectangle (2,30 60x28), "%i", text variable: m_Input_BALAYAGE.PRM_NbBal, invisible if: NOT Global_Variables.PRG_USER.ACTU_USER.MAINTENANCE OR NOT MACHINE.STATE_Manu, input disabled if: (m_Input_BALAYAGE.STATE_LOC) <> 0
        OnMouseDown: write the text variable via InputWithLimits, min 1, max 8
    RoundedRectangle (164,33 52x23), "ON", invisible if: NOT m_Input_BALAYAGE.STATE_ON
    RoundedRectangle (164,33 52x23), "OFF", invisible if: NOT m_Input_BALAYAGE.STATE_OFF
    RoundedRectangle (128,5 87x23), "REMOTE", invisible if: not m_Input_BALAYAGE.OUT_RMT
    RoundedRectangle (128,5 87x23), "LOCAL", invisible if: m_Input_BALAYAGE.OUT_RMT
    RoundedRectangle (107,33 52x23), "RDY", colour toggle: (m_Input_BALAYAGE.STATE_RDY) <> 0
    Rectangle (126,3 91x27), invisible if: Not m_Input_BALAYAGE.AUTOR_Remote_IHM, input disabled if: NOT PRG_User.ACTU_USER.MAINTENANCE
        tap m_Input_BALAYAGE.M_Remote
END_VISUALIZATION

// ---- Visualizations/Symbole/EVAP/VISU_SWEEP_CHEETAH.TcVIS
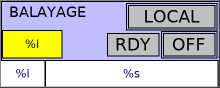
VISUALIZATION VISU_SWEEP_CHEETAH  // 220x88
VAR_IN_OUT
	m_Input_BALAYAGE : BLOCK_TELEMARK_CHEETAH_SWEEP;
END_VAR
    Rectangle (0,0 220x88)
    Rectangle (6,1 117x22), "BALAYAGE"
    Rectangle (0,60 45x27), "%i", text variable: m_Input_BALAYAGE.STATE_NbBal
    Rectangle (45,60 173x27), "%s", text variable: m_Input_BALAYAGE.STATE_BAL
    RoundedRectangle (2,30 60x28), "%i", text variable: m_Input_BALAYAGE.PRM_NbBal, invisible if: NOT Global_Variables.PRG_USER.ACTU_USER.MAINTENANCE OR NOT MACHINE.STATE_Manu, input disabled if: (m_Input_BALAYAGE.STATE_LOC) <> 0
        OnMouseDown: write the text variable via InputWithLimits, min 1, max 8
    RoundedRectangle (163,33 52x23), "ON", invisible if: NOT m_Input_BALAYAGE.STATE_ON
    RoundedRectangle (163,33 52x23), "OFF", invisible if: NOT m_Input_BALAYAGE.STATE_OFF
    RoundedRectangle (128,5 87x23), "REMOTE", invisible if: not m_Input_BALAYAGE.OUT_RMT
    RoundedRectangle (128,5 87x23), "LOCAL", invisible if: m_Input_BALAYAGE.OUT_RMT
    RoundedRectangle (107,33 52x23), "RDY", colour toggle: (m_Input_BALAYAGE.STATE_RDY) <> 0
    Rectangle (126,3 91x27), invisible if: Not m_Input_BALAYAGE.AUTOR_Remote_IHM, input disabled if: NOT PRG_User.ACTU_USER.MAINTENANCE
        tap m_Input_BALAYAGE.M_Remote
    Rectangle (161,31 56x27), invisible if: Not m_Input_BALAYAGE.AUTOR_Balayage_IHM, input disabled if: NOT PRG_User.ACTU_USER.MAINTENANCE
        tap m_Input_BALAYAGE.M_Balayage
END_VISUALIZATION

// ---- Visualizations/Symbole/EVAP/VISU_XTAL.TcVIS
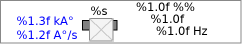
VISUALIZATION VISU_XTAL  // 242x44
VAR_IN_OUT
	m_Input_XTAL : BLOCK_XTAL;
END_VAR
    Rectangle (1,14 85x14), "%1.3f kA°", text variable: m_Input_XTAL.STATE_THICKNESS
    Rectangle (81,3 36x16), "%s", text variable: m_Input_XTAL.MNEMO
    Rectangle (82,20 35x10)
    RoundedRectangle (92,28 17x7)
    Rectangle (121,0 86x14), "%1.0f %%", text variable: m_Input_XTAL.STATE_Life
    Rectangle (120,24 120x14), "%1.0f Hz", text variable: m_Input_XTAL.STATE_FREQUENCY
    Rectangle (121,12 89x14), "%1.0f", text variable: m_Input_XTAL.STATE_ACTIVITY
    Rectangle (3,28 85x14), "%1.2f A°/s", text variable: m_Input_XTAL.STATE_RATE
    Image (89,18 24x23), invisible if: NOT m_Input_XTAL.STATE_NOK, image: MesImages.warning
END_VISUALIZATION

// ---- Visualizations/Symbole/EVAP/VISU_XTAL6_ZOOM.TcVIS
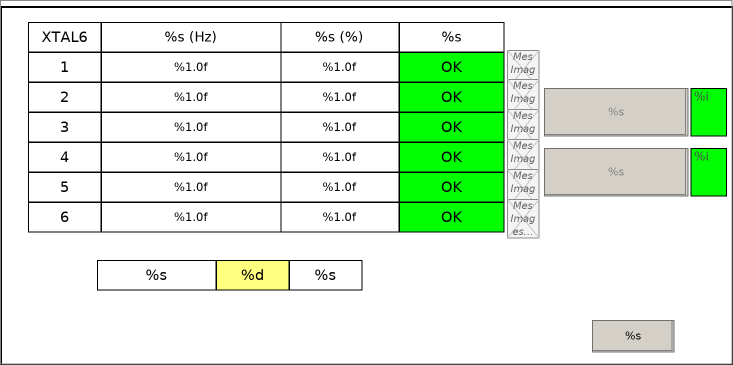
VISUALIZATION VISU_XTAL6_ZOOM  // 733x365, background image fond_blanc_1280_1024
VAR_IN_OUT
	m_Input_XTAL6 : BLOCK_XTAL6;
END_VAR
    Rectangle (0,6 733x359)
    RoundedRectangle (280,52 119x30), "%1.0f", text variable: m_Input_XTAL6.STATE_LIFE[1]
    RoundedRectangle (280,82 119x30), "%1.0f", text variable: m_Input_XTAL6.STATE_LIFE[2]
    RoundedRectangle (280,112 119x30), "%1.0f", text variable: m_Input_XTAL6.STATE_LIFE[3]
    RoundedRectangle (28,52 73x30), "1"
    RoundedRectangle (28,82 73x30), "2"
    RoundedRectangle (28,112 73x30), "3"
    RoundedRectangle (280,22 119x30), "%s (%)", text list: 'TextList_IC6', text index: 13
    RoundedRectangle (399,22 105x30), "%s", text list: 'TextList_IC6', text index: 14
    RoundedRectangle (399,52 105x30), "FAIL", invisible if: NOT m_Input_XTAL6.STATE_QF1
    RoundedRectangle (399,52 105x30), "OK", invisible if: (m_Input_XTAL6.STATE_QF1) <> 0
    RoundedRectangle (399,82 105x30), "FAIL", invisible if: NOT m_Input_XTAL6.STATE_QF2
    RoundedRectangle (399,82 105x30), "OK", invisible if: (m_Input_XTAL6.STATE_QF2) <> 0
    RoundedRectangle (399,112 105x30), "FAIL", invisible if: NOT m_Input_XTAL6.STATE_QF3
    RoundedRectangle (399,112 105x30), "OK", invisible if: (m_Input_XTAL6.STATE_QF3) <> 0
    RoundedRectangle (280,142 119x30), "%1.0f", text variable: m_Input_XTAL6.STATE_LIFE[4]
    RoundedRectangle (280,172 119x30), "%1.0f", text variable: m_Input_XTAL6.STATE_LIFE[5]
    RoundedRectangle (280,202 119x30), "%1.0f", text variable: m_Input_XTAL6.STATE_LIFE[6]
    RoundedRectangle (28,142 73x30), "4"
    RoundedRectangle (28,172 73x30), "5"
    RoundedRectangle (28,202 73x30), "6"
    RoundedRectangle (399,142 105x30), "FAIL", invisible if: NOT m_Input_XTAL6.STATE_QF4
    RoundedRectangle (399,142 105x30), "OK", invisible if: (m_Input_XTAL6.STATE_QF4) <> 0
    RoundedRectangle (399,172 105x30), "FAIL", invisible if: NOT m_Input_XTAL6.STATE_QF5
    RoundedRectangle (399,172 105x30), "OK", invisible if: (m_Input_XTAL6.STATE_QF5) <> 0
    RoundedRectangle (399,202 105x30), "FAIL", invisible if: NOT m_Input_XTAL6.STATE_QF6
    RoundedRectangle (399,202 105x30), "OK", invisible if: (m_Input_XTAL6.STATE_QF6) <> 0
    RoundedRectangle (28,22 73x30), "XTAL6"
    RoundedRectangle (97,260 119x30), "%s", text list: 'TextList_SA_Operations', text index: 23
    RoundedRectangle (216,260 73x30), "%d", text variable: m_Input_XTAL6.PRM_CONS_POSITION_QZ, input disabled if: NOT Global_Variables.PRG_USER.ACTU_USER.MAINTENANCE OR MACHINE.STATE_Prod
        OnMouseDown: write the text variable via VisuDialogs.Numpad, min 1, max 6
    RoundedRectangle (289,260 73x30), "%s", text variable: m_Input_XTAL6.STATE_POSITION
    RoundedRectangle (101,52 180x30), "%1.0f", text variable: m_Input_XTAL6.STATE_FREQUENCY[1]
    RoundedRectangle (101,82 180x30), "%1.0f", text variable: m_Input_XTAL6.STATE_FREQUENCY[2]
    RoundedRectangle (101,112 180x30), "%1.0f", text variable: m_Input_XTAL6.STATE_FREQUENCY[3]
    RoundedRectangle (101,22 180x30), "%s (Hz)", text list: 'TextList_IC6', text index: 12
    RoundedRectangle (101,142 180x30), "%1.0f", text variable: m_Input_XTAL6.STATE_FREQUENCY[4]
    RoundedRectangle (101,172 180x30), "%1.0f", text variable: m_Input_XTAL6.STATE_FREQUENCY[5]
    RoundedRectangle (101,202 180x30), "%1.0f", text variable: m_Input_XTAL6.STATE_FREQUENCY[6]
    Image (507,50 32x39), invisible if: NOT m_Input_XTAL6.ALM_SURV_ACTIVITY_QZ1.DEF AND NOT m_Input_XTAL6.ALM_SURV_LIFE_QZ1.DEF, image: MesImages.warning
    Image (507,79 32x39), invisible if: NOT m_Input_XTAL6.ALM_SURV_ACTIVITY_QZ2.DEF AND NOT m_Input_XTAL6.ALM_SURV_LIFE_QZ2.DEF, image: MesImages.warning
    Image (507,109 32x39), invisible if: NOT m_Input_XTAL6.ALM_SURV_ACTIVITY_QZ3.DEF AND NOT m_Input_XTAL6.ALM_SURV_LIFE_QZ3.DEF, image: MesImages.warning
    Image (507,139 32x39), invisible if: NOT m_Input_XTAL6.ALM_SURV_ACTIVITY_QZ4.DEF AND NOT m_Input_XTAL6.ALM_SURV_LIFE_QZ4.DEF, image: MesImages.warning
    Image (507,169 32x39), invisible if: NOT m_Input_XTAL6.ALM_SURV_ACTIVITY_QZ5.DEF AND NOT m_Input_XTAL6.ALM_SURV_LIFE_QZ5.DEF, image: MesImages.warning
    Image (507,199 32x39), invisible if: NOT m_Input_XTAL6.ALM_SURV_ACTIVITY_QZ6.DEF AND NOT m_Input_XTAL6.ALM_SURV_LIFE_QZ6.DEF, image: MesImages.warning
    Frame (544,88 185x50)
        shows VISU_FCTS_SA(m_Input_ID_XML := 21, m_Input_Operation := m_Input_XTAL6.OP_Scan_Quartz, m_Input_UserRight := PRG_USER.ACTU_USER.FONCTION_SA AND NOT MACHINE.STATE_PROD)
    Frame (544,148 185x50)
        shows VISU_FCTS_SA(m_Input_ID_XML := 22, m_Input_Operation := m_Input_XTAL6.OP_Positionnement, m_Input_UserRight := PRG_USER.ACTU_USER.FONCTION_SA AND NOT MACHINE.STATE_PROD)
    Button (592,320 82x32), "%s", text list: 'TextList_Basiques', text index: 8
        OnMouseClick: change screen: Previous 
        OnMouseClick: execute { .VISU_INDEX_MANU := 0; }
END_VISUALIZATION

// ---- Visualizations/Symbole/EVAP/VISU_XTAL6_PROD.TcVIS
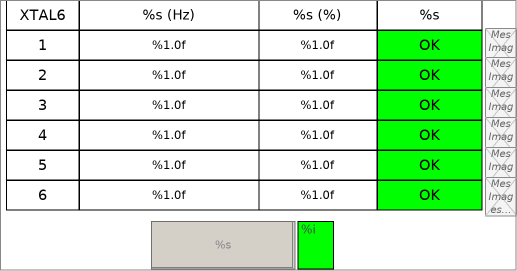
VISUALIZATION VISU_XTAL6_PROD  // 517x271, background image fond_blanc_1280_1024
VAR_IN_OUT
	m_Input_XTAL6 : BLOCK_XTAL6;
END_VAR
    RoundedRectangle (258,30 119x30), "%1.0f", text variable: m_Input_XTAL6.STATE_LIFE[1]
    RoundedRectangle (258,60 119x30), "%1.0f", text variable: m_Input_XTAL6.STATE_LIFE[2]
    RoundedRectangle (258,90 119x30), "%1.0f", text variable: m_Input_XTAL6.STATE_LIFE[3]
    RoundedRectangle (6,30 73x30), "1"
    RoundedRectangle (6,60 73x30), "2"
    RoundedRectangle (6,90 73x30), "3"
    RoundedRectangle (258,0 119x30), "%s (%)", text list: 'TextList_IC6', text index: 13
    RoundedRectangle (377,0 105x30), "%s", text list: 'TextList_IC6', text index: 14
    RoundedRectangle (377,30 105x30), "FAIL", invisible if: NOT m_Input_XTAL6.STATE_QF1
    RoundedRectangle (377,30 105x30), "OK", invisible if: (m_Input_XTAL6.STATE_QF1) <> 0
    RoundedRectangle (377,60 105x30), "FAIL", invisible if: NOT m_Input_XTAL6.STATE_QF2
    RoundedRectangle (377,60 105x30), "OK", invisible if: (m_Input_XTAL6.STATE_QF2) <> 0
    RoundedRectangle (377,90 105x30), "FAIL", invisible if: NOT m_Input_XTAL6.STATE_QF3
    RoundedRectangle (377,90 105x30), "OK", invisible if: (m_Input_XTAL6.STATE_QF3) <> 0
    RoundedRectangle (258,120 119x30), "%1.0f", text variable: m_Input_XTAL6.STATE_LIFE[4]
    RoundedRectangle (258,150 119x30), "%1.0f", text variable: m_Input_XTAL6.STATE_LIFE[5]
    RoundedRectangle (258,180 119x30), "%1.0f", text variable: m_Input_XTAL6.STATE_LIFE[6]
    RoundedRectangle (6,120 73x30), "4"
    RoundedRectangle (6,150 73x30), "5"
    RoundedRectangle (6,180 73x30), "6"
    RoundedRectangle (377,120 105x30), "FAIL", invisible if: NOT m_Input_XTAL6.STATE_QF4
    RoundedRectangle (377,120 105x30), "OK", invisible if: (m_Input_XTAL6.STATE_QF4) <> 0
    RoundedRectangle (377,150 105x30), "FAIL", invisible if: NOT m_Input_XTAL6.STATE_QF5
    RoundedRectangle (377,150 105x30), "OK", invisible if: (m_Input_XTAL6.STATE_QF5) <> 0
    RoundedRectangle (377,180 105x30), "FAIL", invisible if: NOT m_Input_XTAL6.STATE_QF6
    RoundedRectangle (377,180 105x30), "OK", invisible if: (m_Input_XTAL6.STATE_QF6) <> 0
    RoundedRectangle (6,0 73x30), "XTAL6"
    RoundedRectangle (79,30 180x30), "%1.0f", text variable: m_Input_XTAL6.STATE_FREQUENCY[1]
    RoundedRectangle (79,60 180x30), "%1.0f", text variable: m_Input_XTAL6.STATE_FREQUENCY[2]
    RoundedRectangle (79,90 180x30), "%1.0f", text variable: m_Input_XTAL6.STATE_FREQUENCY[3]
    RoundedRectangle (79,0 180x30), "%s (Hz)", text list: 'TextList_IC6', text index: 12
    RoundedRectangle (79,120 180x30), "%1.0f", text variable: m_Input_XTAL6.STATE_FREQUENCY[4]
    RoundedRectangle (79,150 180x30), "%1.0f", text variable: m_Input_XTAL6.STATE_FREQUENCY[5]
    RoundedRectangle (79,180 180x30), "%1.0f", text variable: m_Input_XTAL6.STATE_FREQUENCY[6]
    Image (485,28 32x39), invisible if: NOT m_Input_XTAL6.ALM_SURV_ACTIVITY_QZ1.DEF AND NOT m_Input_XTAL6.ALM_SURV_LIFE_QZ1.DEF, image: MesImages.warning
    Image (485,57 32x39), invisible if: NOT m_Input_XTAL6.ALM_SURV_ACTIVITY_QZ2.DEF AND NOT m_Input_XTAL6.ALM_SURV_LIFE_QZ2.DEF, image: MesImages.warning
    Image (485,87 32x39), invisible if: NOT m_Input_XTAL6.ALM_SURV_ACTIVITY_QZ3.DEF AND NOT m_Input_XTAL6.ALM_SURV_LIFE_QZ3.DEF, image: MesImages.warning
    Image (485,117 32x39), invisible if: NOT m_Input_XTAL6.ALM_SURV_ACTIVITY_QZ4.DEF AND NOT m_Input_XTAL6.ALM_SURV_LIFE_QZ4.DEF, image: MesImages.warning
    Image (485,147 32x39), invisible if: NOT m_Input_XTAL6.ALM_SURV_ACTIVITY_QZ5.DEF AND NOT m_Input_XTAL6.ALM_SURV_LIFE_QZ5.DEF, image: MesImages.warning
    Image (485,177 32x39), invisible if: NOT m_Input_XTAL6.ALM_SURV_ACTIVITY_QZ6.DEF AND NOT m_Input_XTAL6.ALM_SURV_LIFE_QZ6.DEF, image: MesImages.warning
    Frame (151,221 185x50)
        shows VISU_FCTS_SA(m_Input_ID_XML := 21, m_Input_Operation := m_Input_XTAL6.OP_Scan_Quartz, m_Input_UserRight := PRG_USER.ACTU_USER.FONCTION_SA AND NOT MACHINE.STATE_PROD)
END_VISUALIZATION

// ---- Visualizations/Symbole/EVAP/VISU_XTAL_6.TcVIS
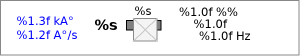
VISUALIZATION VISU_XTAL_6  // 300x56
VAR_IN_OUT
	m_Input_XTAL : BLOCK_XTAL6;
END_VAR

VAR_INPUT
	m_Input_NumFrame_Manu:	USINT;		(*numéro de frame à afficher dans le synoptique MANUEL*)
END_VAR
    Rectangle (0,0 300x56)
        OnMouseClick: execute { .VISU_INDEX_MANU := m_Input_NumFrame_Manu; }
        OnMouseClick: change screen: SYN_MANUEL
    Rectangle (1,14 85x14), "%1.3f kA°", text variable: m_Input_XTAL.STATE_THICKNESS
    Rectangle (125,3 36x16), "%s", text variable: m_Input_XTAL.MNEMO
    Rectangle (126,20 35x10)
    RoundedRectangle (136,28 17x7)
    Rectangle (164,5 86x14), "%1.0f %%", text variable: m_Input_XTAL.STATE_ACTUAL_CRYS_LIFE
    Rectangle (163,29 120x14), "%1.0f Hz", text variable: m_Input_XTAL.STATE_ACTUAL_CRYS_FREQ
    Rectangle (164,17 89x14), "%1.0f", text variable: m_Input_XTAL.STATE_ACTUAL_CRYS_ACTIVITY
    Rectangle (3,28 85x14), "%1.2f A°/s", text variable: m_Input_XTAL.STATE_RATE
    Image (133,18 24x23), invisible if: NOT m_Input_XTAL.STATE_NOK, image: MesImages.warning
    Rectangle (86,16 40x18), "%s", text variable: m_Input_XTAL.STATE_POSITION
END_VISUALIZATION

// ---- Visualizations/Symbole/GAZ/VISU_CONFIG_LIGNE_GAZ_SEUIL.TcVIS
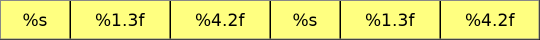
VISUALIZATION VISU_CONFIG_LIGNE_GAZ_SEUIL  // 540x40
VAR_IN_OUT
	m_Input_MASSFLOW:		BLOCK_MFC_BROOKS_NoCoE;
END_VAR
    Rectangle (70,0 100x40), "%1.3f", text variable: m_Input_MASSFLOW.CONF_Nom_Coef, input disabled if: NOT Global_Variables.PRG_USER.ACTU_USER.CONF_MACHINE
        OnMouseDown: write the text variable via InputWithLimits
    Rectangle (170,0 100x40), "%4.2f", text variable: m_Input_MASSFLOW.CONF_Nom_max_flow, input disabled if: NOT Global_Variables.PRG_USER.ACTU_USER.CONF_MACHINE
        OnMouseDown: write the text variable via InputWithLimits
    Rectangle (340,0 100x40), "%1.3f", text variable: m_Input_MASSFLOW.CONF_Util_Coef, input disabled if: NOT Global_Variables.PRG_USER.ACTU_USER.CONF_MACHINE
        OnMouseDown: write the text variable via InputWithLimits
    Rectangle (440,0 100x40), "%4.2f", text variable: m_Input_MASSFLOW.CONF_Util_Max_Flow, input disabled if: NOT Global_Variables.PRG_USER.ACTU_USER.CONF_MACHINE
    Rectangle (0,0 70x40), "%s", text variable: m_Input_MASSFLOW.CONF_Nom_Name, input disabled if: NOT Global_Variables.PRG_USER.ACTU_USER.CONF_MACHINE
        OnMouseDown: write the text variable via InputWithLimits
    Rectangle (270,0 70x40), "%s", text variable: m_Input_MASSFLOW.CONF_Util_Name, input disabled if: NOT Global_Variables.PRG_USER.ACTU_USER.CONF_MACHINE
        OnMouseDown: write the text variable via InputWithLimits
END_VISUALIZATION

// ---- Visualizations/Symbole/GAZ/VISU_CONFIG_LIGNE_GAZ_SEUIL_MFC_MKS.TcVIS
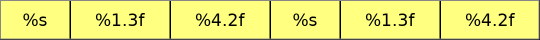
VISUALIZATION VISU_CONFIG_LIGNE_GAZ_SEUIL_MFC_MKS  // 540x40
VAR_IN_OUT
	m_Input_MASSFLOW:		BLOCK_MFC_MKS_NoCoE;
END_VAR
    Rectangle (70,0 100x40), "%1.3f", text variable: m_Input_MASSFLOW.CONF_Nom_Coef, input disabled if: NOT Global_Variables.PRG_USER.ACTU_USER.CONF_MACHINE
        OnMouseDown: write the text variable via Edit
    Rectangle (170,0 100x40), "%4.2f", text variable: m_Input_MASSFLOW.CONF_Nom_max_flow, input disabled if: NOT Global_Variables.PRG_USER.ACTU_USER.CONF_MACHINE
        OnMouseDown: write the text variable via VisuDialogs.Numpad
    Rectangle (340,0 100x40), "%1.3f", text variable: m_Input_MASSFLOW.CONF_Util_Coef, input disabled if: NOT Global_Variables.PRG_USER.ACTU_USER.CONF_MACHINE
        OnMouseDown: write the text variable via VisuDialogs.Numpad
    Rectangle (440,0 100x40), "%4.2f", text variable: m_Input_MASSFLOW.CONF_Util_Max_Flow, input disabled if: NOT Global_Variables.PRG_USER.ACTU_USER.CONF_MACHINE
    Rectangle (0,0 70x40), "%s", text variable: m_Input_MASSFLOW.CONF_Nom_Name, input disabled if: NOT Global_Variables.PRG_USER.ACTU_USER.CONF_MACHINE
        OnMouseDown: write the text variable via VisuDialogs.Keypad
    Rectangle (270,0 70x40), "%s", text variable: m_Input_MASSFLOW.CONF_Util_Name, input disabled if: NOT Global_Variables.PRG_USER.ACTU_USER.CONF_MACHINE
        OnMouseDown: write the text variable via VisuDialogs.Keypad
END_VISUALIZATION

// ---- Visualizations/Symbole/GAZ/VISU_CONFIG_LIGNE_GAZ_SURV.TcVIS
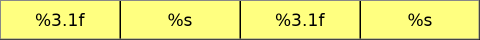
VISUALIZATION VISU_CONFIG_LIGNE_GAZ_SURV  // 480x40
VAR_IN_OUT
	m_Input_MASSFLOW:		BLOCK_MFC_BROOKS_NoCoE;
END_VAR
    Rectangle (0,0 120x40), "%3.1f", text variable: m_Input_MASSFLOW.VAR_ALM_SURV.OFFSET, input disabled if: NOT Global_Variables.PRG_USER.ACTU_USER.CONF_MACHINE
        OnMouseDown: write the text variable via InputWithLimits
    Rectangle (240,0 120x40), "%3.1f", text variable: m_Input_MASSFLOW.VAR_DEF_SURV.offset, input disabled if: NOT Global_Variables.PRG_USER.ACTU_USER.CONF_MACHINE
        OnMouseDown: write the text variable via InputWithLimits
    Rectangle (120,0 120x40), "%s", text variable: m_Input_MASSFLOW.ALM_SURV.delay, input disabled if: NOT Global_Variables.PRG_USER.ACTU_USER.CONF_MACHINE
        OnMouseDown: write the text variable via InputWithLimits
    Rectangle (360,0 120x40), "%s", text variable: m_Input_MASSFLOW.DEF_SURV.DELAY, input disabled if: NOT Global_Variables.PRG_USER.ACTU_USER.CONF_MACHINE
        OnMouseDown: write the text variable via InputWithLimits
END_VISUALIZATION

// ---- Visualizations/Symbole/GAZ/VISU_CONFIG_LIGNE_GAZ_SURV_MFC_MKS.TcVIS
